// TwinCAT 3 PLC project PLK
// ProgramVersion: 3.1.4024.0
// libraries:
//   Tc2_Standard, * (Beckhoff Automation GmbH)
//   Tc2_System, * (Beckhoff Automation GmbH)
//   Tc3_Module, * (Beckhoff Automation GmbH)
// project tree:
//   DUTs/ Item.TcDUT, Location.TcDUT, Recipe.TcDUT
//   GVLs/ GVL.TcGVL, LocalVariables.TcGVL
//   / PlcTask.TcTTO
//   POUs/ ActiveLogic.TcPOU, Automatic.TcPOU, BeltLogic.TcPOU, ErrorsWarnings.TcPOU, MAIN.TcPOU, Manual.TcPOU, Motor.TcPOU, PistonInputLogic.TcPOU, PistonOutputLogic.TcPOU, TableLogic.TcPOU, TrackingLogic.TcPOU
// real-time tasks:
//   TASK PlcTask: cycle T#10ms, priority 20, ADS port 350
//   TASK PlcTask1: cycle T#10ms, priority 21, ADS port 351
//   TASK PlcTask2: cycle T#10ms, priority 22, ADS port 352
// I/O:
//   DEVICE Device 1 (EtherCAT), AmsNetId 5.132.85.195.2.1
//     Term 1 (EK1200) [EK1200-7000 EtherCAT Power supply (1,5A E-Bus)]
//       Term 2 (EL1859) [EL1859 8Ch. Dig. Input 24V, 3ms, 8Ch. Dig. Output 24V, 0.5A]
//       Term 3 (EL1859) [EL1859 8Ch. Dig. Input 24V, 3ms, 8Ch. Dig. Output 24V, 0.5A]
//       Term 4 (EL9011) [EL9011 End Terminal]
//   DEVICE Device 2 (NOV-DP-RAM)
//   DEVICE Device 3 (CX7000), AmsNetId 5.132.85.195.4.1
//     Term 1 (CX7028) [CX7028-0000-0118]
//       modules: Module 1 (DIO_2x), Module 3 (DIO_2x), Module 5 (DI_2x), Module 7 (DI_2x)
// variable links:
//   PLK/PLK Instance <-> Device 1 (EtherCAT)/Term 1 (EK1200)/Term 2 (EL1859)
//     PlcTask Inputs/GVL.FotocellInput <-> Channel 1/Input
//     PlcTask Inputs/GVL.FotocellOutput <-> Channel 6/Input
//     PlcTask Inputs/GVL.SwitchCompressor <-> Channel 3/Input
//     PlcTask Inputs/GVL.SwitchPress <-> Channel 2/Input
//     PlcTask Inputs/GVL.SwitchTableExit <-> Channel 5/Input
//     PlcTask Inputs/GVL.SwitchTablePosition <-> Channel 4/Input
//     PlcTask Outputs/GVL.MotorCompressor <-> Channel 9/Output
//     PlcTask Outputs/GVL.MotorTableDirection <-> Channel 13/Output
//     PlcTask Outputs/GVL.MotorTableMove <-> Channel 14/Output
//     PlcTask Outputs/GVL.PistonInputBackwards <-> Channel 11/Output
//     PlcTask Outputs/GVL.PistonInputForward <-> Channel 10/Output
//     PlcTask Outputs/GVL.PistonOutputBackwards <-> Channel 15/Output
//     PlcTask Outputs/GVL.PistonOutputForward <-> Channel 16/Output
//     PlcTask Outputs/GVL.PistonPress <-> Channel 12/Output
//   PLK/PLK Instance <-> Device 1 (EtherCAT)/Term 1 (EK1200)/Term 3 (EL1859)
//     PlcTask Outputs/GVL.MotorBeltDirection <-> Channel 9/Output
//     PlcTask Outputs/GVL.MotorBeltMove <-> Channel 10/Output
//   PLK/PLK Instance <-> Device 3 (CX7000)/Term 1 (CX7028)
//     PlcTask Inputs/GVL.ButtonBLB <-> Module 5 (DI_2x)/DI_2x Input Channel 1/Input
//     PlcTask Inputs/GVL.ButtonBLT <-> Module 1 (DIO_2x)/DIO_2x Inputs Channel 2/Input
//     PlcTask Inputs/GVL.ButtonBRB <-> Module 5 (DI_2x)/DI_2x Input Channel 2/Input
//     PlcTask Inputs/GVL.ButtonBRT <-> Module 3 (DIO_2x)/DIO_2x Input Channel 1/Input
//     PlcTask Inputs/GVL.ButtonGreen <-> Module 3 (DIO_2x)/DIO_2x Input Channel 2/Input
//     PlcTask Inputs/GVL.ButtonRed <-> Module 1 (DIO_2x)/DIO_2x Inputs Channel 1/Input
//     PlcTask Inputs/GVL.Switch <-> Module 7 (DI_2x)/DI_2x Inputs Channel 1/Input
//     PlcTask Outputs/GVL.LEDBlueBottom <-> Module 3 (DIO_2x)/DIO_2x Outputs Channel 2/Output
//     PlcTask Outputs/GVL.LEDBlueTop <-> Module 1 (DIO_2x)/DIO_2x Outputs Channel 2/Output
//     PlcTask Outputs/GVL.LEDGreen <-> Module 3 (DIO_2x)/DIO_2x Outputs Channel 1/Output
//     PlcTask Outputs/GVL.LEDRed <-> Module 1 (DIO_2x)/DIO_2x Outputs Channel 1/Output

CONFIGURATION PLK
    RESOURCE PLC ON TwinCAT3
        TASK PlcTask(INTERVAL := T#10ms, PRIORITY := 22);
        PROGRAM MAIN WITH PlcTask : MAIN;
    END_RESOURCE
END_CONFIGURATION

// ---- DUTs/Item.TcDUT
TYPE Item :
STRUCT
	Id: UDINT := 0;
	Recipe: Recipe;
END_STRUCT
END_TYPE

// ---- DUTs/Location.TcDUT
TYPE Location :
STRUCT
	Item: Item;
	Active: BOOL;
END_STRUCT
END_TYPE

// ---- DUTs/Recipe.TcDUT
TYPE Recipe :
STRUCT
	WorkingTime: TIME; 
END_STRUCT
END_TYPE

// ---- GVLs/GVL.TcGVL
{attribute 'qualified_only'}
VAR_GLOBAL
	ButtonRed AT %I*: BOOL;
	ButtonBRT AT %I*: BOOL;
	ButtonBLB AT %I*: BOOL;
	Switch AT %I*: BOOL;
	ButtonBLT AT %I*: BOOL;
	ButtonGreen AT %I*: BOOL;
	ButtonBRB AT %I*: BOOL;
	LEDRed AT %Q*: BOOL;
	LEDGreen AT %Q*: BOOL;
	LEDBlueTop AT %Q*: BOOL;
	LEDBlueBottom AT %Q*: BOOL;
	FotocellInput AT %I*: BOOL;
	FotocellOutput AT %I*: BOOL;
	SwitchPress AT %I*: BOOL;
	SwitchTableExit AT %I*: BOOL;
	SwitchTablePosition AT %I*: BOOL;
	SwitchCompressor AT %I*: BOOL;
	MotorCompressor AT %Q*: BOOL;
	MotorTableMove AT %Q*: BOOL;
	MotorTableDirection AT %Q*: BOOL;
	MotorBeltMove AT %Q*: BOOL;
	MotorBeltDirection AT %Q*: BOOL;
	PistonInputForward AT %Q*: BOOL;
	PistonInputBackwards AT %Q*: BOOL;
	PistonPress AT %Q*: BOOL;
	PistonOutputBackwards AT %Q*: BOOL;
	PistonOutputForward AT %Q*: BOOL;
END_VAR

// ---- GVLs/LocalVariables.TcGVL
{attribute 'qualified_only'}
VAR_GLOBAL
	Locations: ARRAY[1..6] OF Location;
	Recipe: Recipe := (WorkingTime := TIME#2s0ms);
END_VAR

// ---- POUs/MAIN.TcPOU
PROGRAM MAIN
VAR
	manual: Manual;
	automatic: Automatic;
	errorsAndWarnings: ErrorsWarnings;
	trackingLogic: TrackingLogic;
	activeLogic: ActiveLogic;
END_VAR

IF gvl.ButtonGreen THEN
	gvl.MotorCompressor := TRUE;
ELSIF gvl.ButtonRed THEN
	gvl.MotorCompressor := FALSE;
END_IF

IF gvl.Switch THEN
	manual();
else
	automatic();
END_IF
trackingLogic();
activeLogic();
errorsAndWarnings();

END_PROGRAM

// ---- POUs/Manual.TcPOU
FUNCTION_BLOCK Manual
VAR
	Counter: CTUD;
	MotorTable: Motor;
	MotorBelt: Motor;
	Backwards: BOOL;
END_VAR

Counter();

gvl.PistonInputBackwards := TRUE;
gvl.PistonInputForward := FALSE;

gvl.MotorTableMove := FALSE;

gvl.PistonPress := FALSE;

gvl.PistonOutputBackwards := TRUE;
gvl.PistonOutputForward := FALSE;

gvl.MotorBeltMove := FALSE;
IF (gvl.ButtonBLT AND Counter.CV > 0) THEN
	Counter.CD := TRUE;
ELSE
	Counter.CD := FALSE;
END_IF


IF (gvl.ButtonBRT AND Counter.CV < 4) THEN
	Counter.CU := TRUE;
ELSE
	Counter.CU := FALSE;
END_IF

IF Counter.CV = 0 THEN
	IF gvl.ButtonBLB THEN
		gvl.PistonInputBackwards := FALSE;
		gvl.PistonInputForward := TRUE;
	ELSE
		gvl.PistonInputBackwards := TRUE;
		gvl.PistonInputForward := FALSE;
	END_IF
	
ELSIF Counter.CV = 1 THEN
	MotorTable(
		Forwards := gvl.ButtonBRB,
		Backwards := gvl.ButtonBLB,
		blockTime := T#0.5S,
		Active => gvl.MotorTableMove,
		Direction => gvl.MotorTableDirection
	);	
	
ELSIF Counter.CV = 2 THEN
	IF gvl.ButtonBLB THEN
		gvl.PistonPress := TRUE;
	ELSE
		gvl.PistonPress := FALSE;
	END_IF
	
ELSIF Counter.CV = 3 THEN
	IF gvl.ButtonBLB THEN
		gvl.PistonOutputBackwards := FALSE;
		gvl.PistonOutputForward := TRUE;
	ELSE
		gvl.PistonOutputBackwards := TRUE;
		gvl.PistonOutputForward := FALSE;
	END_IF
	
ELSIF Counter.CV = 4 THEN
	MotorBelt(
		Forwards := gvl.ButtonBRB,
		Backwards := gvl.ButtonBLB,
		blockTime := T#0.5S,
		Active => gvl.MotorBeltMove,
		Direction => gvl.MotorBeltDirection
	);
END_IF

END_FUNCTION_BLOCK

// ---- POUs/Motor.TcPOU
FUNCTION_BLOCK Motor
VAR_OUTPUT
	Direction: BOOL;
	Active: BOOL;
END_VAR
VAR_INPUT
	Forwards: BOOL;
	Backwards: BOOL;
	blockTime: TIME;
END_VAR
VAR
	timerForward: TOF;
	timerBackward: TOF;
	blockForward: BOOL;
	blockBackward: BOOL;
	rotateForward: BOOL;
	rotateBackward: BOOL;
	fallTrigForward: F_TRIG;
	fallDetectedForward: BOOL;
	fallTrigBackward: F_TRIG;
	fallDetectedBackward: BOOL;
END_VAR

fallTrigForward(CLK := Forwards, Q => fallDetectedForward);
fallTrigBackward(CLK := Backwards, Q => fallDetectedBackward);

timerForward(IN := fallDetectedForward, PT := blockTime, Q => blockBackward);
timerBackward(IN := fallDetectedBackward, PT := blockTime, Q => blockForward);

rotateForward := Forwards AND NOT blockForward;
rotateBackward := Backwards AND NOT blockBackward;


IF rotateForward OR rotateBackward THEN
	IF rotateForward THEN
		Direction := TRUE;
	ELSIF rotateBackward THEN 
		Direction := FALSE;
	END_IF
	
	Active := TRUE;
ELSE
	Active := FALSE;
END_IF

END_FUNCTION_BLOCK

// ---- POUs/Automatic.TcPOU
FUNCTION_BLOCK Automatic
VAR_INPUT
END_VAR
VAR_OUTPUT
END_VAR
VAR
	inputPiston: PistonInputLogic;
	outputPiston: PistonOutputLogic;
	tableLogic: TableLogic;
	beltLogic: BeltLogic;
END_VAR

inputPiston();
tableLogic();
outputPiston();
beltLogic();

END_FUNCTION_BLOCK

// ---- POUs/PistonInputLogic.TcPOU
FUNCTION_BLOCK PistonInputLogic
VAR
	timer: TOF;
	timerElapsed: BOOL;
	counter: CTU;
	id: UDINT;
	item: Item;
	location: Location;
END_VAR

timer(IN :=  NOT gvl.FotocellInput AND gvl.SwitchTablePosition, PT := T#1S, Q => timerElapsed);
//counter();

IF timerElapsed AND LocalVariables.Locations[2].Item.Id = 0 THEN
	gvl.PistonInputBackwards := FALSE;
	gvl.PistonInputForward := TRUE;
//	LocalVariables.Locations[2].Item.Id := LocalVariables.Locations[1].Item.Id;
//	LocalVariables.Locations[2].Item.Recipe := LocalVariables.Locations[1].Item.Recipe;
	
//ELSIF NOT gvl.FotocellInput THEN
//	counter.CU := TRUE;
//	id := counter.CV;
//	LocalVariables.Locations[1].Item.Id := id;
//	LocalVariables.Locations[1].Item.Recipe := LocalVariables.Recipe;

ELSE
	gvl.PistonInputBackwards := TRUE;
	gvl.PistonInputForward := FALSE;
	//counter.CU := FALSE;
	//LocalVariables.Locations[1].Item.Id := NULL;
END_IF

END_FUNCTION_BLOCK

// ---- POUs/PistonOutputLogic.TcPOU
FUNCTION_BLOCK PistonOutputLogic
VAR
	timer: TOF;
	timerElapsed: BOOL;
	riseTrig: R_TRIG;
	riseTrigDetected: BOOL;
END_VAR

timer(IN := gvl.SwitchTableExit, PT := T#0.5S, Q => timerElapsed);
//riseTrig(CLK := gvl.SwitchTableExit, Q => riseTrigDetected);

IF timerElapsed THEN
	gvl.PistonOutputBackwards := FALSE;
	gvl.PistonOutputForward := TRUE;
	gvl.MotorBeltMove := TRUE;
ELSE
	gvl.PistonOutputBackwards := TRUE;
	gvl.PistonOutputForward := FALSE;
END_IF

//IF riseTrigDetected THEN
//	LocalVariables.Locations[5].Item.Id := LocalVariables.Locations[4].Item.Id;
//	LocalVariables.Locations[5].Item.Recipe := LocalVariables.Locations[4].Item.Recipe;
//	LocalVariables.Locations[4].Item.Id := NULL;
//	LocalVariables.Locations[4].Item.Recipe := LocalVariables.Recipe;
//END_IF

END_FUNCTION_BLOCK

// ---- POUs/TableLogic.TcPOU
FUNCTION_BLOCK TableLogic
VAR
	timer: TOF;
	timerElapsed: BOOL;
	riseTrig: R_TRIG;
	riseTrigDetected: BOOL;
	fallTrig: F_TRIG;
	fallTrigDetected: BOOL;
END_VAR

riseTrig(CLK := gvl.SwitchPress, Q => riseTrigDetected);
//fallTrig(CLK:= gvl.SwitchPress, Q => fallTrigDetected);
timer(IN := riseTrigDetected, PT := LocalVariables.Recipe.WorkingTime, Q => timerElapsed);
gvl.MotorTableMove := TRUE;

//IF riseTrigDetected THEN
//	LocalVariables.Locations[3].Item.Id := LocalVariables.Locations[2].Item.Id;
//	LocalVariables.Locations[3].Item.Recipe := LocalVariables.Locations[2].Item.Recipe;
//	LocalVariables.Locations[2].Item.Id := NULL;
//	LocalVariables.Locations[2].Item.Recipe := LocalVariables.Recipe;
//END_IF

IF timerElapsed THEN
	gvl.PistonPress := TRUE;
	gvl.MotorTableMove := FALSE;
ELSIF NOT gvl.FotocellOutput THEN
	gvl.MotorTableMove := FALSE;
	gvl.PistonPress := FALSE;
ELSE	
	gvl.PistonPress := FALSE;
	gvl.MotorTableMove := TRUE;
END_IF

//IF fallTrigDetected THEN
//	LocalVariables.Locations[4].Item.Id := LocalVariables.Locations[3].Item.Id;
//	LocalVariables.Locations[4].Item.Recipe := LocalVariables.Locations[3].Item.Recipe;
//	LocalVariables.Locations[3].Item.Id := NULL;
//	LocalVariables.Locations[3].Item.Recipe := LocalVariables.Recipe;
//END_IF

END_FUNCTION_BLOCK

// ---- POUs/BeltLogic.TcPOU
FUNCTION_BLOCK BeltLogic
VAR_INPUT
END_VAR
VAR_OUTPUT
END_VAR
VAR
	fallTrig: F_TRIG;
	fallTrigDetected: bool;
END_VAR

fallTrig(CLK:= gvl.FotocellOutput, Q => fallTrigDetected);

IF NOT LocalVariables.Locations[5].Item.Id = 0 THEN
	gvl.MotorBeltMove := TRUE;
ELSIF NOT gvl.FotocellOutput THEN
	gvl.MotorBeltMove := FALSE;
//ELSIF gvl.FotocellOutput THEN
//	LocalVariables.Locations[6].Item.Id := NULL;
//	LocalVariables.Locations[6].Item.Recipe := LocalVariables.Recipe;
END_IF

//IF fallTrigDetected THEN
//	LocalVariables.Locations[6].Item.Id := LocalVariables.Locations[5].Item.Id;
//	LocalVariables.Locations[6].Item.Recipe := LocalVariables.Locations[5].Item.Recipe;
//	LocalVariables.Locations[5].Item.Id := NULL;
//	LocalVariables.Locations[5].Item.Recipe := LocalVariables.Recipe;
//END_IF

END_FUNCTION_BLOCK

// ---- POUs/ErrorsWarnings.TcPOU
FUNCTION_BLOCK ErrorsWarnings
VAR_INPUT
END_VAR
VAR_OUTPUT
END_VAR
VAR
	CompressorNotRunning: BOOL;
	LineBackedUp: BOOL;
	BeltWrongDirection: BOOL;
	TableWrongDirection: BOOL;
END_VAR

// ERRORS
CompressorNotRunning := NOT gvl.MotorCompressor;
	

//WARNINGS
LineBackedUp := NOT gvl.FotocellOutput;
BeltWrongDirection := gvl.MotorBeltDirection;
TableWrongDirection := gvl.MotorTableDirection;

END_FUNCTION_BLOCK

// ---- POUs/TrackingLogic.TcPOU
FUNCTION_BLOCK TrackingLogic
VAR
	timerPistonInput: TOF;
	timerElapsedPistonInput: BOOL;
	counter: CTU;
	id: UDINT;
	item: Item;
	location: Location;
	timerTable: TOF;
	timerElapsedTable: BOOL;
	riseTrigTable: R_TRIG;
	riseTrigDetectedTable: BOOL;
	fallTrigTable: F_TRIG;
	fallTrigDetectedTable: BOOL;
	riseTrigPistonOutput: R_TRIG;
	riseTrigDetectedPistonOutput: BOOL;
	fallTrigBelt: F_TRIG;
	fallTrigDetectedBelt: bool;
	fallTrigPistonInput: F_TRIG;
	fallTrigDetectedPistonInput: BOOL;
END_VAR

//Piston Input logic
timerPistonInput(IN :=  NOT gvl.FotocellInput AND gvl.SwitchTablePosition, PT := T#1S, Q => timerElapsedPistonInput);
fallTrigPistonInput(CLK := gvl.PistonInputForward, Q => fallTrigDetectedPistonInput);
counter();
IF fallTrigDetectedPistonInput AND LocalVariables.Locations[2].Item.Id = 0 THEN
	LocalVariables.Locations[2].Item.Id := LocalVariables.Locations[1].Item.Id;
	LocalVariables.Locations[2].Item.Recipe := LocalVariables.Locations[1].Item.Recipe;
	LocalVariables.Locations[1].Item.Id := NULL;
ELSIF NOT gvl.FotocellInput THEN
	counter.CU := TRUE;
	id := counter.CV;
	LocalVariables.Locations[1].Item.Id := id;
	LocalVariables.Locations[1].Item.Recipe := LocalVariables.Recipe;
ELSE
	counter.CU := FALSE;
END_IF

//Table logic
riseTrigTable(CLK := gvl.SwitchPress, Q => riseTrigDetectedTable);
fallTrigTable(CLK:= gvl.SwitchPress, Q => fallTrigDetectedTable);
timerTable(IN := riseTrigDetectedTable, PT := LocalVariables.Recipe.WorkingTime, Q => timerElapsedTable);

IF riseTrigDetectedTable THEN
	LocalVariables.Locations[3].Item.Id := LocalVariables.Locations[2].Item.Id;
	LocalVariables.Locations[3].Item.Recipe := LocalVariables.Locations[2].Item.Recipe;
	LocalVariables.Locations[2].Item.Id := NULL;
	LocalVariables.Locations[2].Item.Recipe := LocalVariables.Recipe;
END_IF

IF fallTrigDetectedTable THEN
	LocalVariables.Locations[4].Item.Id := LocalVariables.Locations[3].Item.Id;
	LocalVariables.Locations[4].Item.Recipe := LocalVariables.Locations[3].Item.Recipe;
	LocalVariables.Locations[3].Item.Id := NULL;
	LocalVariables.Locations[3].Item.Recipe := LocalVariables.Recipe;
END_IF

//Piston Output logic
riseTrigPistonOutput(CLK := gvl.SwitchTableExit, Q => riseTrigDetectedPistonOutput);

IF riseTrigDetectedPistonOutput THEN
	LocalVariables.Locations[5].Item.Id := LocalVariables.Locations[4].Item.Id;
	LocalVariables.Locations[5].Item.Recipe := LocalVariables.Locations[4].Item.Recipe;
	LocalVariables.Locations[4].Item.Id := NULL;
	LocalVariables.Locations[4].Item.Recipe := LocalVariables.Recipe;
END_IF

//Belt logic
fallTrigBelt(CLK:= gvl.FotocellOutput, Q => fallTrigDetectedBelt);

IF gvl.FotocellOutput THEN
	LocalVariables.Locations[6].Item.Id := NULL;
	LocalVariables.Locations[6].Item.Recipe := LocalVariables.Recipe;
END_IF

IF fallTrigDetectedBelt THEN
	LocalVariables.Locations[6].Item.Id := LocalVariables.Locations[5].Item.Id;
	LocalVariables.Locations[6].Item.Recipe := LocalVariables.Locations[5].Item.Recipe;
	LocalVariables.Locations[5].Item.Id := NULL;
	LocalVariables.Locations[5].Item.Recipe := LocalVariables.Recipe;
END_IF

END_FUNCTION_BLOCK

// ---- POUs/ActiveLogic.TcPOU
FUNCTION_BLOCK ActiveLogic
VAR_INPUT
END_VAR
VAR_OUTPUT
END_VAR
VAR
END_VAR

LocalVariables.Locations[1].Active := gvl.PistonInputForward;
LocalVariables.Locations[2].Active := gvl.MotorTableMove;
LocalVariables.Locations[3].Active := gvl.PistonPress;
LocalVariables.Locations[4].Active := gvl.PistonOutputForward;
LocalVariables.Locations[5].Active := gvl.MotorBeltMove;
LocalVariables.Locations[6].Active := NOT gvl.FotocellOutput;

END_FUNCTION_BLOCK
